TYPE ST_HomeInputs :
STRUCT
    DummyRoom : ST_DummyRoomInputs;
END_STRUCT
END_TYPE

(* stored: Version 1.1.0.1
   DUT ST_HomeInputs: Id {caabb78d-9a4b-4cd9-8764-2a0c0407ce3e} *)
